REGION Network 42: Line CIP Valve AV-02.08
   // CIP Supply Line 1 for CIP Line T-02, T03, T04, T09 to Blending
   RUNG wire#powerrail
      Contact( "AlwaysTRUE" )
      wire#w1
      Contact( "T-02.01_DB"."OUT_AV.08" )
      wire#w2
      Coil( "IO_Valve_T02_Chili"."AV-02.08".AUT_OP )
   END_RUNG
   RUNG wire#w1
      Contact( "T-03.01_DB"."OUT_AV.08" )
   END_RUNG wire#w2
   RUNG wire#w1
      Contact( "T-04.01_DB"."OUT_AV.08" )
   END_RUNG wire#w2
   RUNG wire#w1
      Contact( "T-09.01_DB"."OUT_AV.08" )
   END_RUNG wire#w2
   // the same network as SCL:
   "IO_Valve_T02_Chili"."AV-02.08".AUT_OP := "AlwaysTRUE" AND ("T-02.01_DB"."OUT_AV.08" OR "T-03.01_DB"."OUT_AV.08" OR "T-04.01_DB"."OUT_AV.08" OR "T-09.01_DB"."OUT_AV.08");
END_REGION

REGION Network 43: Line CIP Valve AV-05.11
   // CIP Supply Line 1 for CIP Line T-05, T06, T07, T08 to Blending
   RUNG wire#powerrail
      Contact( "AlwaysTRUE" )
      wire#w1
      Contact( "T-05.01_DB"."OUT_AV.11" )
      wire#w2
      Coil( "IO_Valve_T05_Tomato"."AV-05.11".AUT_OP )
   END_RUNG
   RUNG wire#w1
      Contact( "T-06.01_DB"."OUT_AV.11" )
   END_RUNG wire#w2
   RUNG wire#w1
      Contact( "T-07.01_DB"."OUT_AV.11" )
   END_RUNG wire#w2
   RUNG wire#w1
      Contact( "T-08.01_DB"."OUT_AV.11" )
   END_RUNG wire#w2
   // the same network as SCL:
   "IO_Valve_T05_Tomato"."AV-05.11".AUT_OP := "AlwaysTRUE" AND ("T-05.01_DB"."OUT_AV.11" OR "T-06.01_DB"."OUT_AV.11" OR "T-07.01_DB"."OUT_AV.11" OR "T-08.01_DB"."OUT_AV.11");
END_REGION

REGION Network 44: Line ProWater T09 & T10
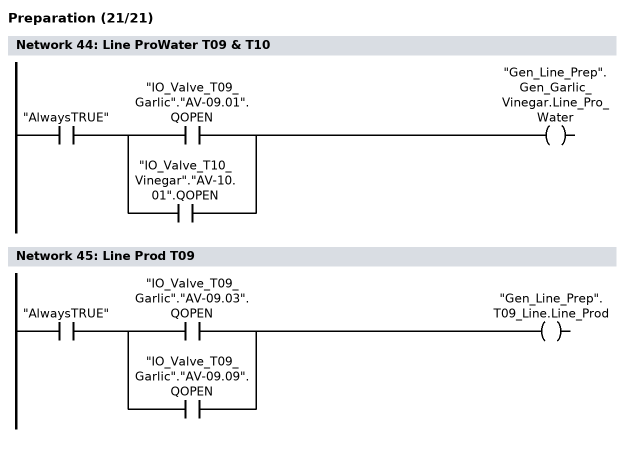
   RUNG wire#powerrail
      Contact( "AlwaysTRUE" )
      wire#w1
      Contact( "IO_Valve_T09_Garlic"."AV-09.01".QOPEN )
      wire#w2
      Coil( "Gen_Line_Prep".Gen_Garlic_Vinegar.Line_Pro_Water )
   END_RUNG
   RUNG wire#w1
      Contact( "IO_Valve_T10_Vinegar"."AV-10.01".QOPEN )
   END_RUNG wire#w2
   // the same network as SCL:
   "Gen_Line_Prep".Gen_Garlic_Vinegar.Line_Pro_Water := "AlwaysTRUE" AND ("IO_Valve_T09_Garlic"."AV-09.01".QOPEN OR "IO_Valve_T10_Vinegar"."AV-10.01".QOPEN);
END_REGION

REGION Network 45: Line Prod T09
   RUNG wire#powerrail
      Contact( "AlwaysTRUE" )
      wire#w1
      Contact( "IO_Valve_T09_Garlic"."AV-09.03".QOPEN )
      wire#w2
      Coil( "Gen_Line_Prep".T09_Line.Line_Prod )
   END_RUNG
   RUNG wire#w1
      Contact( "IO_Valve_T09_Garlic"."AV-09.09".QOPEN )
   END_RUNG wire#w2
   // the same network as SCL:
   "Gen_Line_Prep".T09_Line.Line_Prod := "AlwaysTRUE" AND ("IO_Valve_T09_Garlic"."AV-09.03".QOPEN OR "IO_Valve_T09_Garlic"."AV-09.09".QOPEN);
END_REGION

NETWORK
TITLE = Valve IO
//Valve T-01.01 Hotwater Tank
      CALL  "IO Valve T01 HWT", "IO_Valve_T01_HWT"
      ( lock  := ,
        Init  := "General_DB".Initial,
        Reset := "General_DB".Reset
      );
//Valve T-02.01 Chili Awetan Tank 1
      CALL  "IO Valve T02 Chili", "IO_Valve_T02_Chili"
      ( lock    := ,
        Init    := "General_DB".Initial,
        testing := ,
        Reset   := "General_DB".Reset
      );
//Valve T-03.01 Chili Awetan Tank 2
      CALL  "IO Valve T03 Chili", "IO_Valve_T03_Chili"
      ( lock    := ,
        Init    := "General_DB".Initial,
        testing := ,
        Reset   := "General_DB".Reset
      );
//Valve T-04.01 Chili Awetan Tank 3
      CALL  "IO Valve T04 Chili", "IO_Valve_T04_Chili"
      ( lock    := ,
        Init    := "General_DB".Initial,
        testing := ,
        Reset   := "General_DB".Reset
      );
//Valve T-05.01 Tomato Tank
      CALL  "IO Valve T05 Tomato", "IO_Valve_T05_Tomato"
      ( lock    := ,
        Init    := "General_DB".Initial,
        testing := ,
        Reset   := "General_DB".Reset
      );
//Valve T-06.01 Fresh Chili Tank 1
      CALL  "IO Valve T06 FreshChili", "IO_Valve_T06_FreshChili"
      ( lock    := ,
        Init    := "General_DB".Initial,
        testing := ,
        Reset   := "General_DB".Reset
      );
//Valve T-07.01 Fresh Chili Tank 2
      CALL  "IO Valve T07 FreshChili", "IO_Valve_T07_FreshChili"
      ( lock    := ,
        Init    := "General_DB".Initial,
        testing := ,
        Reset   := "General_DB".Reset
      );
//Valve T-08.01 Fresh Chili Tank 3
      CALL  "IO Valve T08 FreshChili", "IO_Valve_T08_FreshChili"
      ( lock    := ,
        Init    := "General_DB".Initial,
        testing := ,
        Reset   := "General_DB".Reset
      );
//Valve T-09.01 Garlic Tank
      CALL  "IO Valve T09 Garlic", "IO_Valve_T09_Garlic"
      ( lock    := ,
        Init    := "General_DB".Initial,
        testing := ,
        Reset   := "General_DB".Reset
      );
//Valve T-10.01 Vinegar Tank
      CALL  "IO Valve T10 Vinegar", "IO_Valve_T10_Vinegar"
      ( lock    := ,
        Init    := "General_DB".Initial,
        testing := ,
        Reset   := "General_DB".Reset
      );
//Valve T-10.01 Vinegar Tank
      CALL  "IO Valve T51 HotWaterLine", "IO_Valve_T51_HW"
      ( lock    := ,
        Init    := "General_DB".Initial,
        testing := ,
        Reset   := "General_DB".Reset
      );


END_FUNCTION
